(* CoDeSys 2.3 export: PUMP.EXP *)

(* Global variable list: Pump *)
VAR_GLOBAL

	Pump_FlawAutoSet_1:		REAL;
	Pump_FlawAutoSet_2:		REAL;
	Pump_FlawAutoSet_3:		REAL;
	Pump_FlawAutoSet_4:		REAL;



END_VAR
